FUNCTION_BLOCK DELAY_200
VAR_INPUT
	IN : REAL;
	N : INT;
	RST : BOOL;
END_VAR
VAR_OUTPUT
	OUT : REAL;
END_VAR
VAR
	buf : ARRAY[0..199] OF REAL;
	i : INT;
	init: BOOL;
	stop: INT;
END_VAR

(*
version 1.0	10. nov. 2020
programmer 	PhOstmann

this function block delays input values by each programm cycle
after N+1 cycles the in value has shifted to the out.
N can be any alue from 0 .. 200
if n = 0 the input will be present on the output without a delay.
f N > 200 then the output will be delayed by 200 cycles.
any high on rst will load the buffer with in.

*)

stop := LIMIT(0,N,200) - 1;
IF rst OR NOT init THEN
	init := TRUE;
	FOR i := 0 TO stop DO buf[i] := in; END_FOR;
	out := in;
	i := 0;
ELSIF stop < 0 THEN
	out := in;
ELSE
	out := buf[i];
	buf[i] := in;
	i := INC1(i, N);
END_IF;



(* revision history

*)

END_FUNCTION_BLOCK

(* stored: Version 1.1.0.1, ProductVersion 3.1.4024.3
   POU DELAY_200: Id {dccbaad1-090b-4f47-939e-05951b94d60f}, SpecialFunc None *)
